FUNCTION_BLOCK FB_Inputs 
VAR_INPUT
	fbJoystickWinch : FB_JoystickInputScaling; 
	fbJoystickRot : FB_JoystickInputScaling; 
	fbDisplacementSlider : FB_JoystickInputScaling_01;
	fbYokeInputScaling : FB_Yoke_Input_Scaling;
	fbWinchPosition : FB_Encoder;
	fbPressureSupply : FB_PressureInputScaling; 
	fbPressureReturn : FB_PressureInputScaling;
	fbPressureWinch_A_Input : FB_PressureInputScaling;
	fbPressureWInch_B_Input : FB_PressureInputScaling; 
END_VAR
VAR_OUTPUT
END_VAR
VAR
END_VAR

fbJoystickWinch(
	bEnable := G_IO.bAutoSwitch OR G_IO.bManualSwitch,
	nRawInput := G_IO.fJoyYraw, 
	stJoystickInputScaling := G_Parameters.stParam.stJoystickInputScalingY, 
	fNormalizedOutput => G_Sensors.fJoystickNormalizedY
);

fbJoystickRot(
	bEnable := G_IO.bManualSwitch, 
	nRawInput := G_IO.fJoyZraw,
	stJoystickInputScaling := G_Parameters.stParam.stJoystickInputScalingZ,
    fNormalizedOutput => G_Sensors.fJoystickNormalizedZ
);

fbDisplacementSlider(
	bEnable := G_IO.bAutoSwitch OR G_IO.bManualSwitch,
	nRawInput := G_IO.fJoyXraw, 
	stJoystickInputScaling := G_Parameters.stParam.stJoystickInputScalingX, 
	fNormalizedOutput => G_Sensors.fJoystickNormalizedX
);


fbYokeInputScaling(
	bEnable := TRUE, //Vil lese Yokeverdi hele tiden så den settes til TRUE (var G_IO.bManualSwitch før)
	nRawInput := G_IO.fYoke, 
	stYokeInputScaling := G_Parameters.stParam.stYokeInputScaling,
	fNormalizedOutput => G_Sensors.fYokeNormalizedFeedback
);

fbWinchPosition(
nRawInput := G_IO.nWinchEncoderValue,
fEncoderOffset := G_Parameters.stParam.fWinchEncoderOffset,
fPosition => G_Sensors.fWinchEncoderPosition
);

fbPressureSupply(
	nRawInput := G_IO.fPressureSupply,
	stPressureInputScaling := G_Parameters.stParam.stPressureSensorScaling400bar,
	fOutput => G_Sensors.fPressureSupply
);

fbPressureReturn(
	nRawInput := G_IO.fPressureReturn,
	stPressureInputScaling := G_Parameters.stParam.stPressureSensorScaling40bar,
	fOutput => G_Sensors.fPressureReturn
	);
	
fbPressureWinch_A_Input(
	nRawInput := G_IO.fPressureWinchA, 
	stPressureInputScaling := G_Parameters.stParam.stPressureSensorScaling400bar, 
	fOutput => G_Sensors.fPressureWinchA
	);
	
fbPressureWinch_B_Input(
nRawInput := G_IO.fPressureWinchB,
stPressureInputScaling := G_Parameters.stParam.stPressureSensorScaling400bar, 
fOutput => G_Sensors.fPressureWinchB
);

// Trykkfall over motor: 

G_Sensors.fDeltaPMotor := (G_Sensors.fPressureWinchA - G_Sensors.fPressureWinchB);

END_FUNCTION_BLOCK

(* stored: Version 1.1.0.1
   POU FB_Inputs: Id {6a583cfe-140e-4485-b87b-9b85c9186e72}, SpecialFunc None *)
